// SIMATIC S7-200 SMART project (STEP 7-Micro/WIN SMART), CPU ST20

SYMBOL_TABLE 系统符号
Always_On        SM0.0    // 始终接通
END_SYMBOL_TABLE

ORGANIZATION_BLOCK MAIN:OB1
TITLE=程序注释
BEGIN
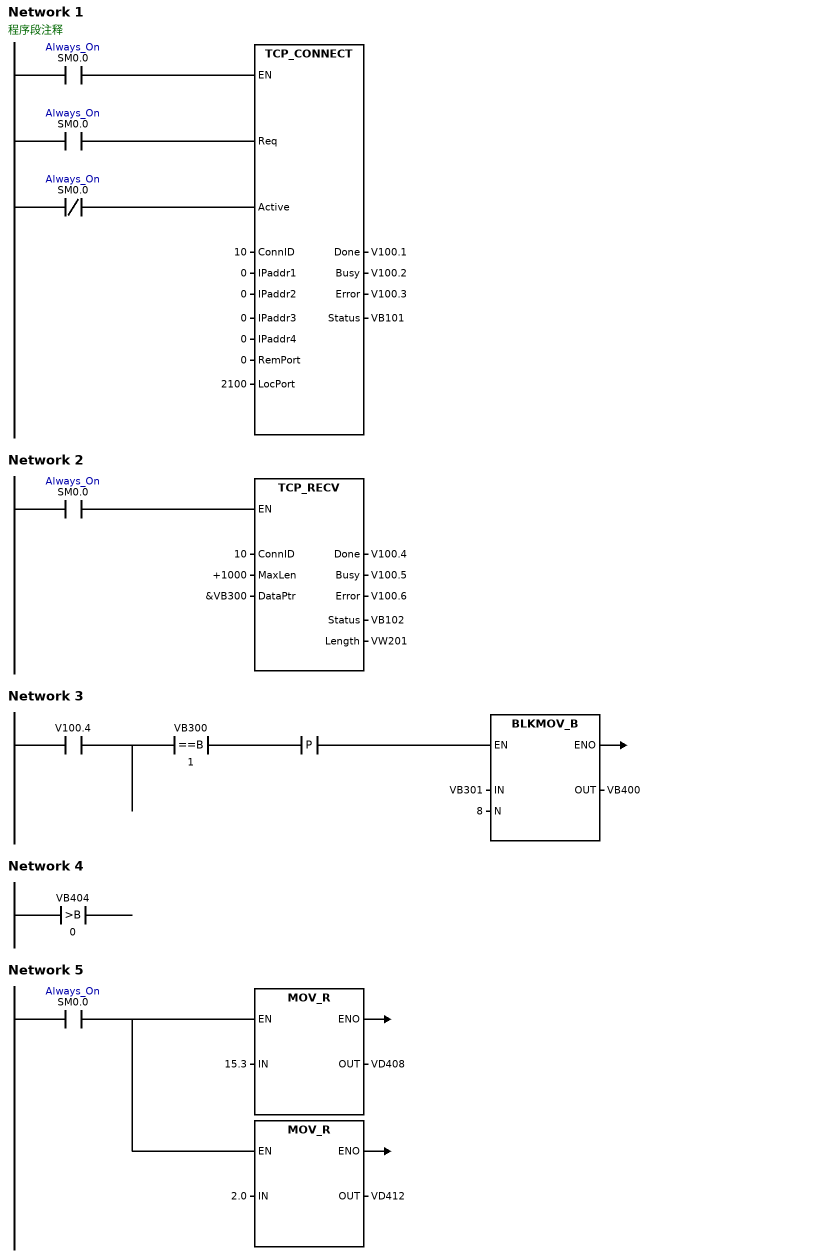
Network 1
// 程序段注释
LD     Always_On:SM0.0
=      L60.0
LD     Always_On:SM0.0
=      L63.7
LDN    Always_On:SM0.0
=      L63.6
LD     L60.0
CALL   TCP_CONNECT:SBR1, L63.7, L63.6, 10, 0, 0, 0, 0, 0, 2100, V100.1, V100.2, V100.3, VB101
Network 2
LD     Always_On:SM0.0
CALL   TCP_RECV:SBR2, 10, +1000, &VB300, V100.4, V100.5, V100.6, VB102, VW201
Network 3
// (network saved uncompiled; LAD cells follow)
// row 0: c0 -| |- V100.4 v  c1 -|==B|- VB300, 1  c2 -|P|-  c3 --  c4 [BLKMOV_B EN:=power@row0, IN:=VB301, N:=8, ENO=>power, OUT=>VB400]  c5 ->
// row 1: c0 ^  c4 [box]
Network 4
// (network saved uncompiled; LAD cells follow)
// row 0: c0 -|>B|- VB404, 0
Network 5
LD     Always_On:SM0.0
MOVR   15.3, VD408
MOVR   2.0, VD412
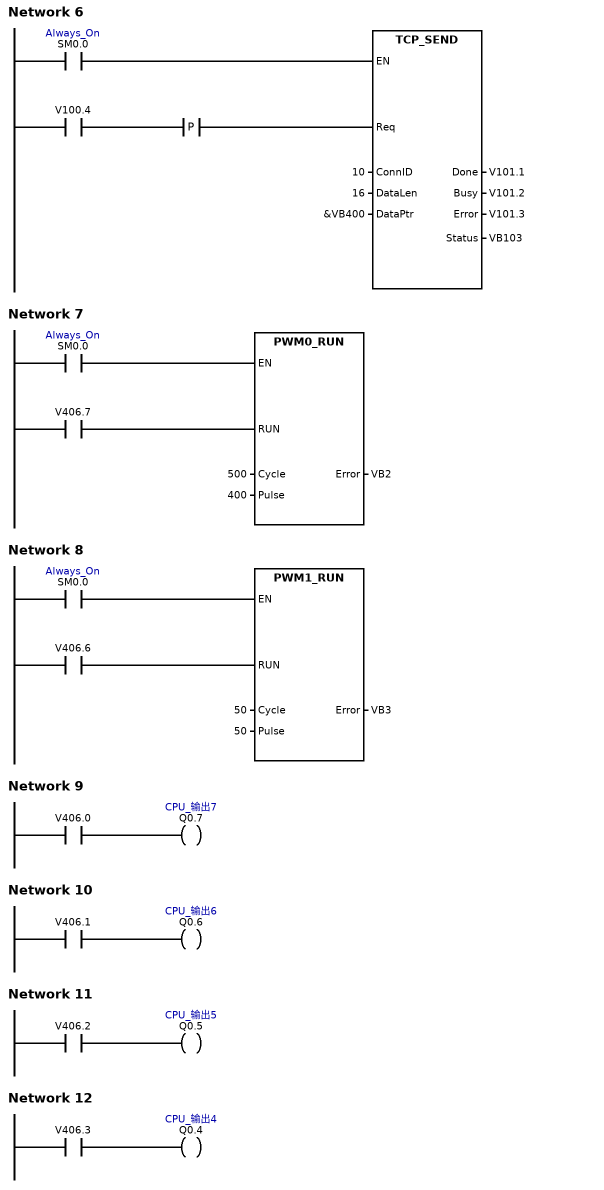
Network 6
LD     Always_On:SM0.0
=      L60.0
LD     V100.4
EU
=      L63.7
LD     L60.0
CALL   TCP_SEND:SBR5, L63.7, 10, 16, &VB400, V101.1, V101.2, V101.3, VB103
Network 7
LD     Always_On:SM0.0
=      L60.0
LD     V406.7
=      L63.7
LD     L60.0
CALL   PWM0_RUN:SBR3, L63.7, 500, 400, VB2
Network 8
LD     Always_On:SM0.0
=      L60.0
LD     V406.6
=      L63.7
LD     L60.0
CALL   PWM1_RUN:SBR4, L63.7, 50, 50, VB3
Network 9
LD     V406.0
=      CPU_输出7:Q0.7
Network 10
LD     V406.1
=      CPU_输出6:Q0.6
Network 11
LD     V406.2
=      CPU_输出5:Q0.5
Network 12
LD     V406.3
=      CPU_输出4:Q0.4
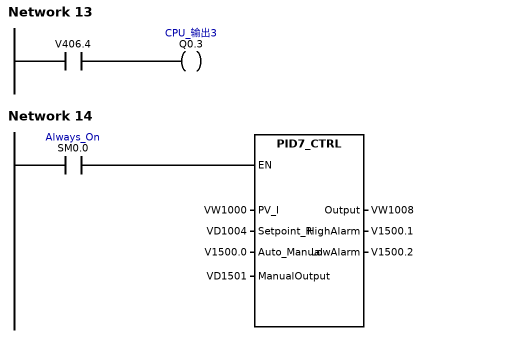
Network 13
LD     V406.4
=      CPU_输出3:Q0.3
Network 14
LD     Always_On:SM0.0
CALL   PID7_CTRL:SBR7, VW1000, VD1004, V1500.0, VD1501, VW1008, V1500.1, V1500.2
END_ORGANIZATION_BLOCK

// SBR1: protected block, not included

// SBR2: protected block, not included

// SBR3: protected block, not included

// SBR4: protected block, not included

// SBR5: protected block, not included

// SBR6: protected block, not included

// SBR7: protected block, not included

// INT1: protected block, not included
